Staubli VAL3: onEdit.pgx

public program onEdit(string& x_sItem[])
  local string l_sItem
begin
  //
  // compose the string
  // call getType(l_sItem)
  // x_sItem=l_sItem+" ???"
  //
end
